Yaskawa INFORM job: pos_y_0.JBI

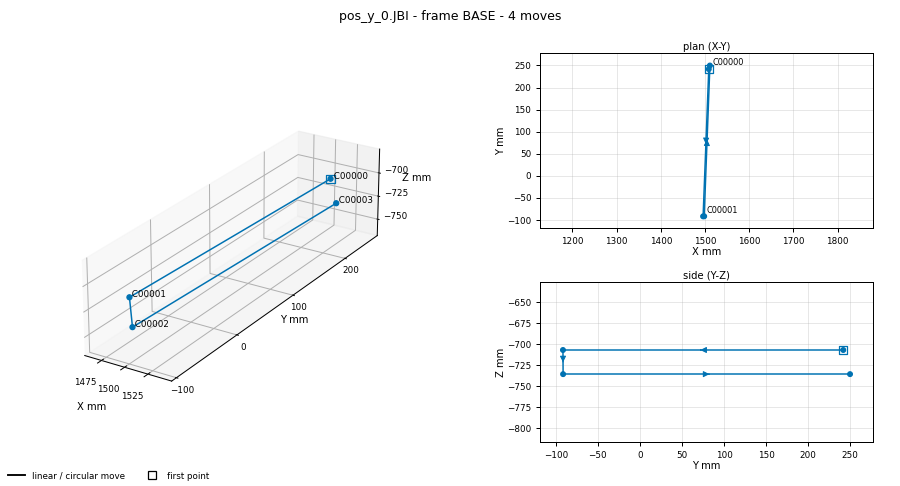
[picture p0: tool path of pos_y_0.JBI in frame BASE, 4 of 6 moves have a stored position in this frame; points joined in program order, loops and branches not executed]
/JOB
//NAME pos_y_0
//POS
///NPOS 4,0,4,0,0,0
///TOOL 0
///POSTYPE BASE
///RECTAN
///RCONF 0,0,0,0,0,0,0,0,0,0,0,0,0,0,0,0,0,0,0,0,0,0,0,0
C00000=1508.548100,241.812870,-706.912550,180.000000,-60.000000,0.000000
C00001=1495.702100,-91.547130,-706.912550,180.000000,-60.000000,0.000000
C00002=1498.155100,-91.387130,-735.628050,180.000000,-60.000000,0.000000
C00003=1511.059100,249.862870,-735.628050,180.000000,-60.000000,0.000000
///POSTYPE PULSE
///PULSE
EX000=184320
///POSTYPE PULSE
///PULSE
EC00000=184320
EC00001=184320
EC00002=184320
EC00003=184320
//INST
///DATE 2023/08/07 14:38
///ATTR SC,RW,RJ
////FRAME BASE
///GROUP1 RB1,ST1
NOP
MOVJ P009 EX000 VJ=15.00
MOVJ C00000 EC00000 VJ=15.0
CALL JOB:SPYON
MOVL C00001 EC00001 V=150.0
MOVL C00002 EC00002 V=150.0
MOVL C00003 EC00003 V=150.0
CALL JOB:SPYOF
MOVJ P009 VJ=15.00
END
